TYPE WordStringUnion :
UNION
	ValWord	: WORD;
	ValString	: STRING;
END_UNION
END_TYPE

(* stored: Version 1.1.0.1, ProductVersion 3.1.4024.11
   DUT WordStringUnion: Id {269e64fa-437e-4f91-80fa-e0ee3febceb6} *)
